PROGRAM PRG_13_MES
VAR
	MesData					: HttpGet;
	tonRecycle01			: TON;
END_VAR

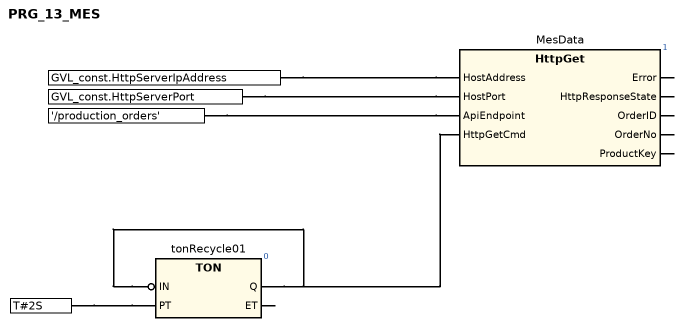
tonRecycle01(IN := NOT tonRecycle01.Q, PT := T#2S); // TON
MesData(
    HostAddress := GVL_const.HttpServerIpAddress,
    HostPort := GVL_const.HttpServerPort,
    ApiEndpoint := '/production_orders',
    HttpGetCmd := tonRecycle01.Q); // HttpGet

END_PROGRAM

(* stored: Version 1.1.0.1, ProductVersion 3.1.4024.15
   POU PRG_13_MES: Id {19557303-94c8-41da-8e4d-a7c8ca793dd0}, SpecialFunc None *)
